FUNCTION_BLOCK FB_SunblindSwitch
VAR_INPUT
	bEn			:BOOL;
	bUp			:BOOL;
	bDwn		:BOOL;
	bPos_steht	:BOOL;
	bSet_Angle	:BOOL;
	nSlid_Pos 	:INT;
	nSlid_Angl 	:INT;
	uiSwiOvrTi	:UDINT;
END_VAR
VAR_OUTPUT
	st_SunBld			: ST_BA_SunBld;
END_VAR
VAR_IN_OUT
	bClicked 	:BOOL;
END_VAR
VAR
	TON_Halten			: TON;
	SR					: SR;
	TON_Dwn_Reset		: TON;
	FB_Value_Change		: FB_Value_Change;
	FB_Value_Change2	: FB_Value_Change;
	FB_Value_Write		: FB_Value_Write;
	FB_Value_Write2		: FB_Value_Write;
	FB_Value_Change_Hys	: FB_Value_Change_Hys;
	FB_Reset			: FB_Reset;
	SR2					: SR;
	TON_Halten2			: TON;
	TON_Up_Reset		: TON;
	tSwiOvrTi			: TIME;

	SR_ManMod: SR;
	TON_Reset_Selbe_Taste_Dwn: TON;
	TON_Reset_Selbe_Taste_Up: TON;
END_VAR
VAR // added by the converter: edge detectors and wires of the graphical bodies
    _w1 : ANY;
    _w2, _w3, _w4, _w5, _w6 : BOOL;
END_VAR

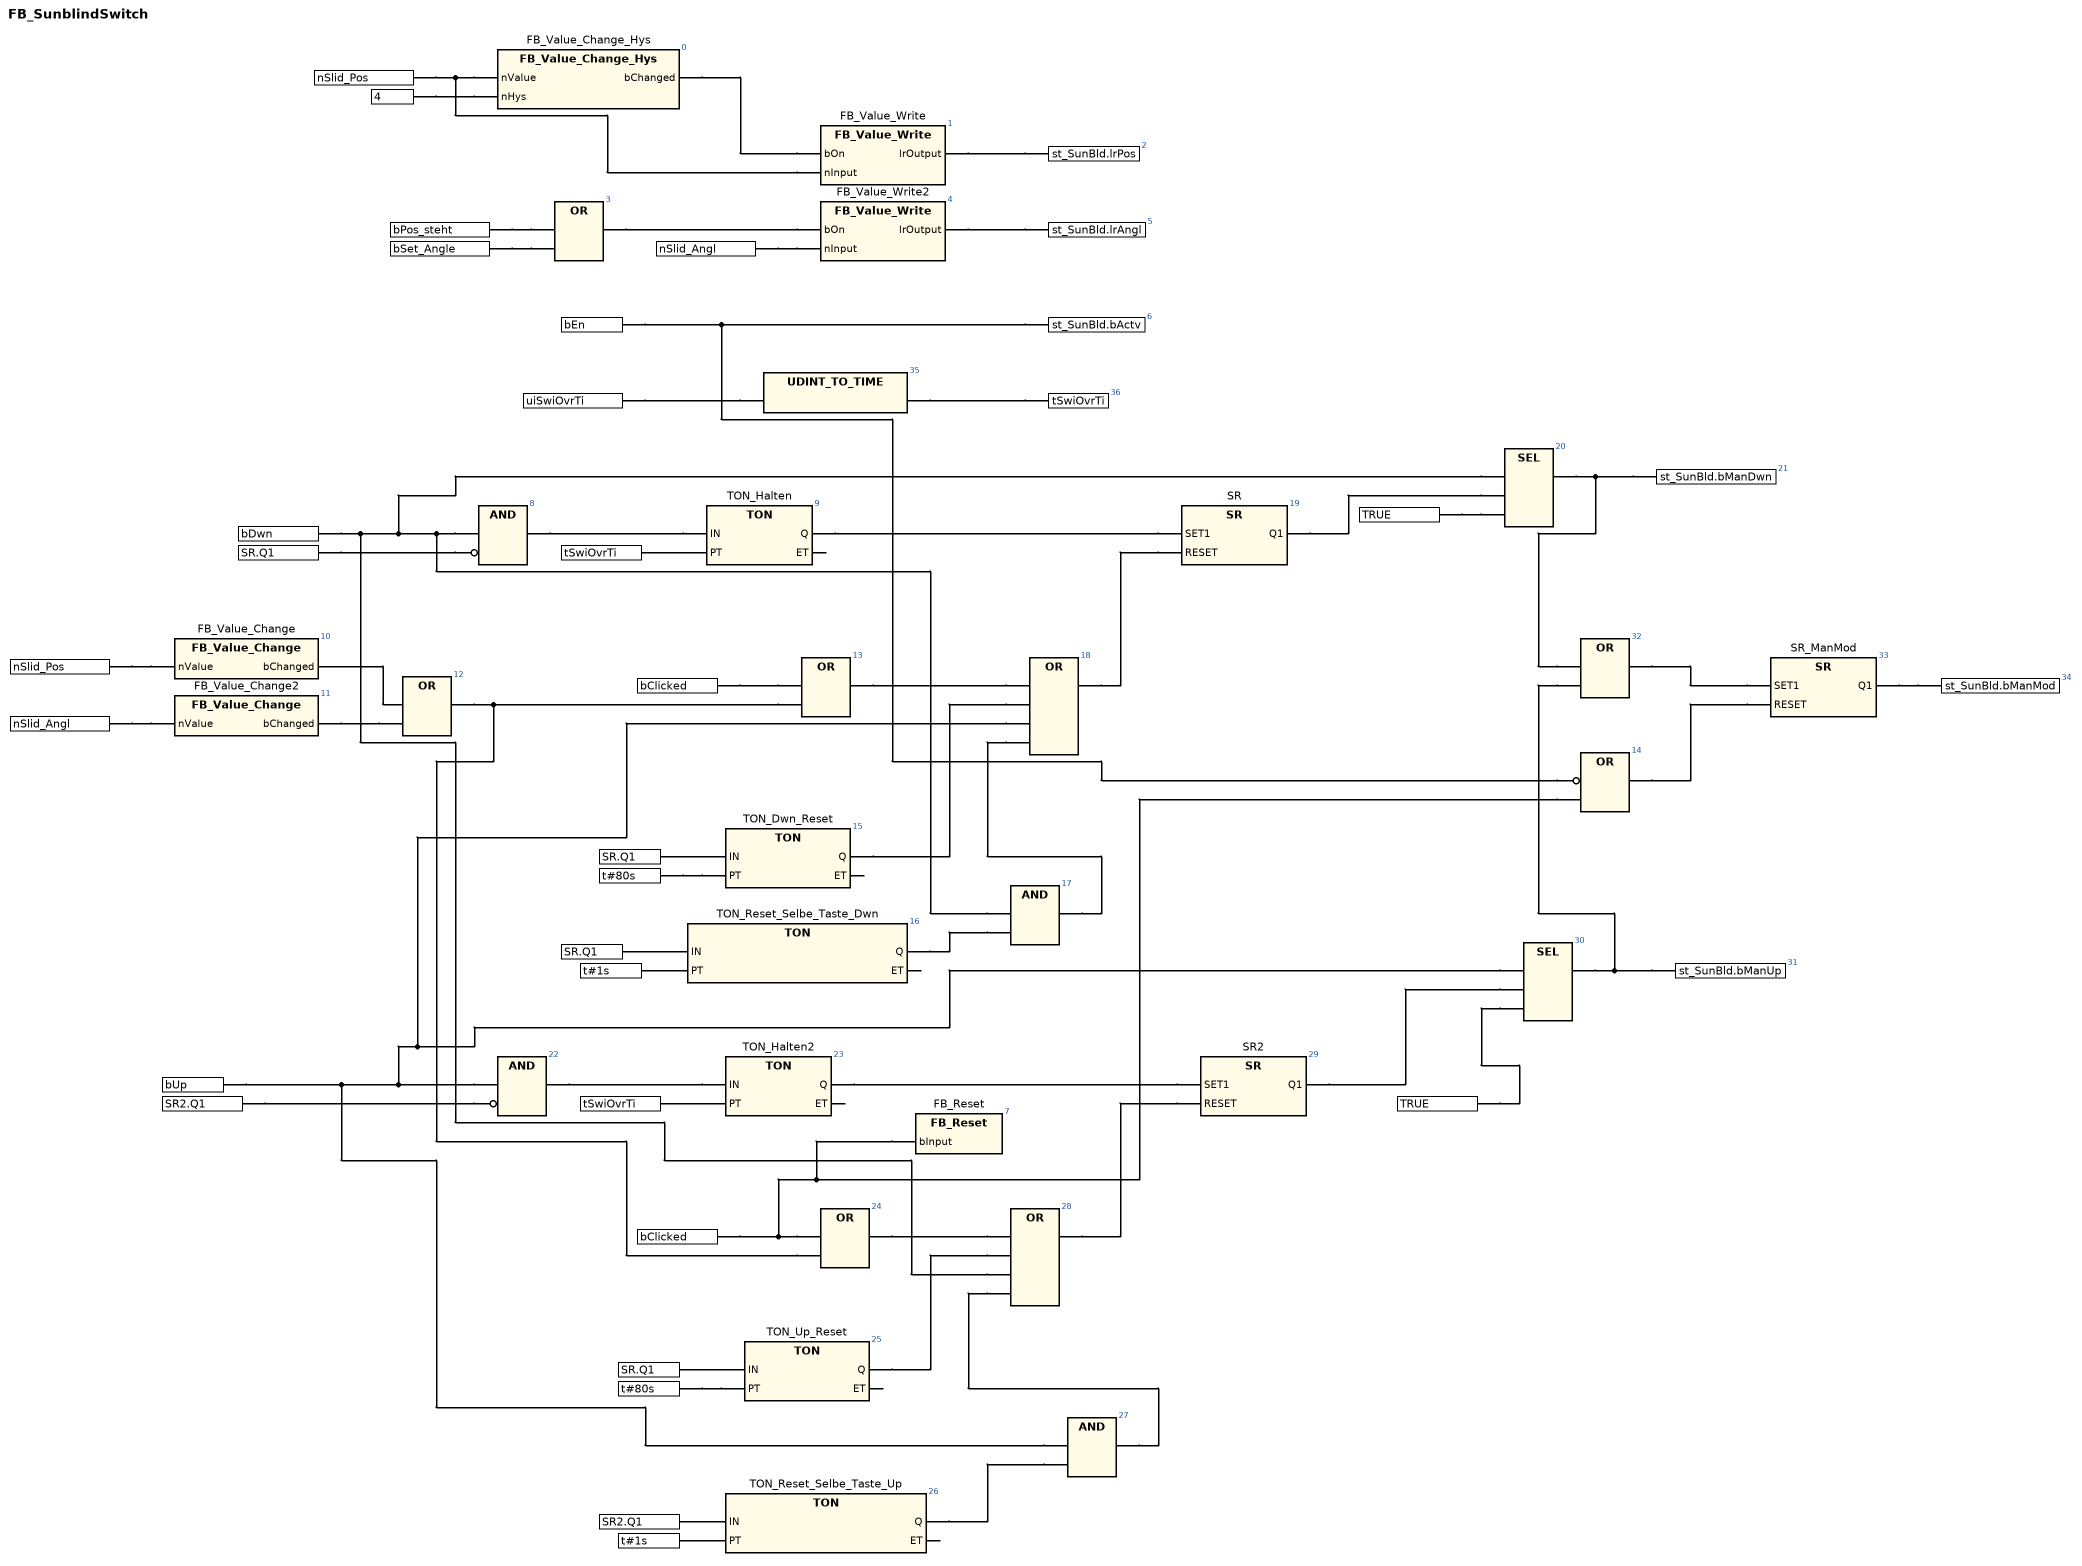
FB_Value_Change_Hys(nValue := nSlid_Pos, nHys := 4);
FB_Value_Write(bOn := FB_Value_Change_Hys.bChanged, nInput := nSlid_Pos);
st_SunBld.lrPos := FB_Value_Write.lrOutput;
FB_Value_Write2(bOn := bPos_steht OR bSet_Angle, nInput := nSlid_Angl); // FB_Value_Write
st_SunBld.lrAngl := FB_Value_Write2.lrOutput;
st_SunBld.bActv := bEn;
FB_Reset(bInput := bClicked);
TON_Halten(IN := bDwn AND NOT SR.Q1, PT := tSwiOvrTi); // TON
FB_Value_Change(nValue := nSlid_Pos);
FB_Value_Change2(nValue := nSlid_Angl); // FB_Value_Change
_w1 := FB_Value_Change.bChanged OR FB_Value_Change2.bChanged;
_w2 := bClicked OR _w1;
_w3 := NOT bEn OR bClicked;
TON_Dwn_Reset(IN := SR.Q1, PT := t#80s); // TON
TON_Reset_Selbe_Taste_Dwn(IN := SR.Q1, PT := t#1s); // TON
SR(SET1 := TON_Halten.Q, RESET := _w2 OR TON_Dwn_Reset.Q OR bUp OR bDwn AND TON_Reset_Selbe_Taste_Dwn.Q);
_w4 := SEL(bDwn, SR.Q1, TRUE);
st_SunBld.bManDwn := _w4;
TON_Halten2(IN := bUp AND NOT SR2.Q1, PT := tSwiOvrTi); // TON
_w5 := bClicked OR _w1;
TON_Up_Reset(IN := SR.Q1, PT := t#80s); // TON
TON_Reset_Selbe_Taste_Up(IN := SR2.Q1, PT := t#1s); // TON
SR2(SET1 := TON_Halten2.Q, RESET := _w5 OR TON_Up_Reset.Q OR bDwn OR bUp AND TON_Reset_Selbe_Taste_Up.Q); // SR
_w6 := SEL(bUp, SR2.Q1, TRUE);
st_SunBld.bManUp := _w6;
SR_ManMod(SET1 := _w4 OR _w6, RESET := _w3); // SR
st_SunBld.bManMod := SR_ManMod.Q1;
tSwiOvrTi := UDINT_TO_TIME(uiSwiOvrTi);

END_FUNCTION_BLOCK

(* stored: Version 1.1.0.1, ProductVersion 3.1.4022.12
   POU FB_SunblindSwitch: Id {dba517b0-d0b6-414e-b8e9-367c0f8d097a}, SpecialFunc None *)
